# EPICS autosave request: iocBoot/iocTomoScan_32IDC/auto_settings.req
file "tomoScan_settings.req", P=$(P), R=$(R)
file "tomoScan_PSO_settings.req", P=$(P), R=$(R)
file "tomoScan_32IDC_settings.req", P=$(P), R=$(R)
